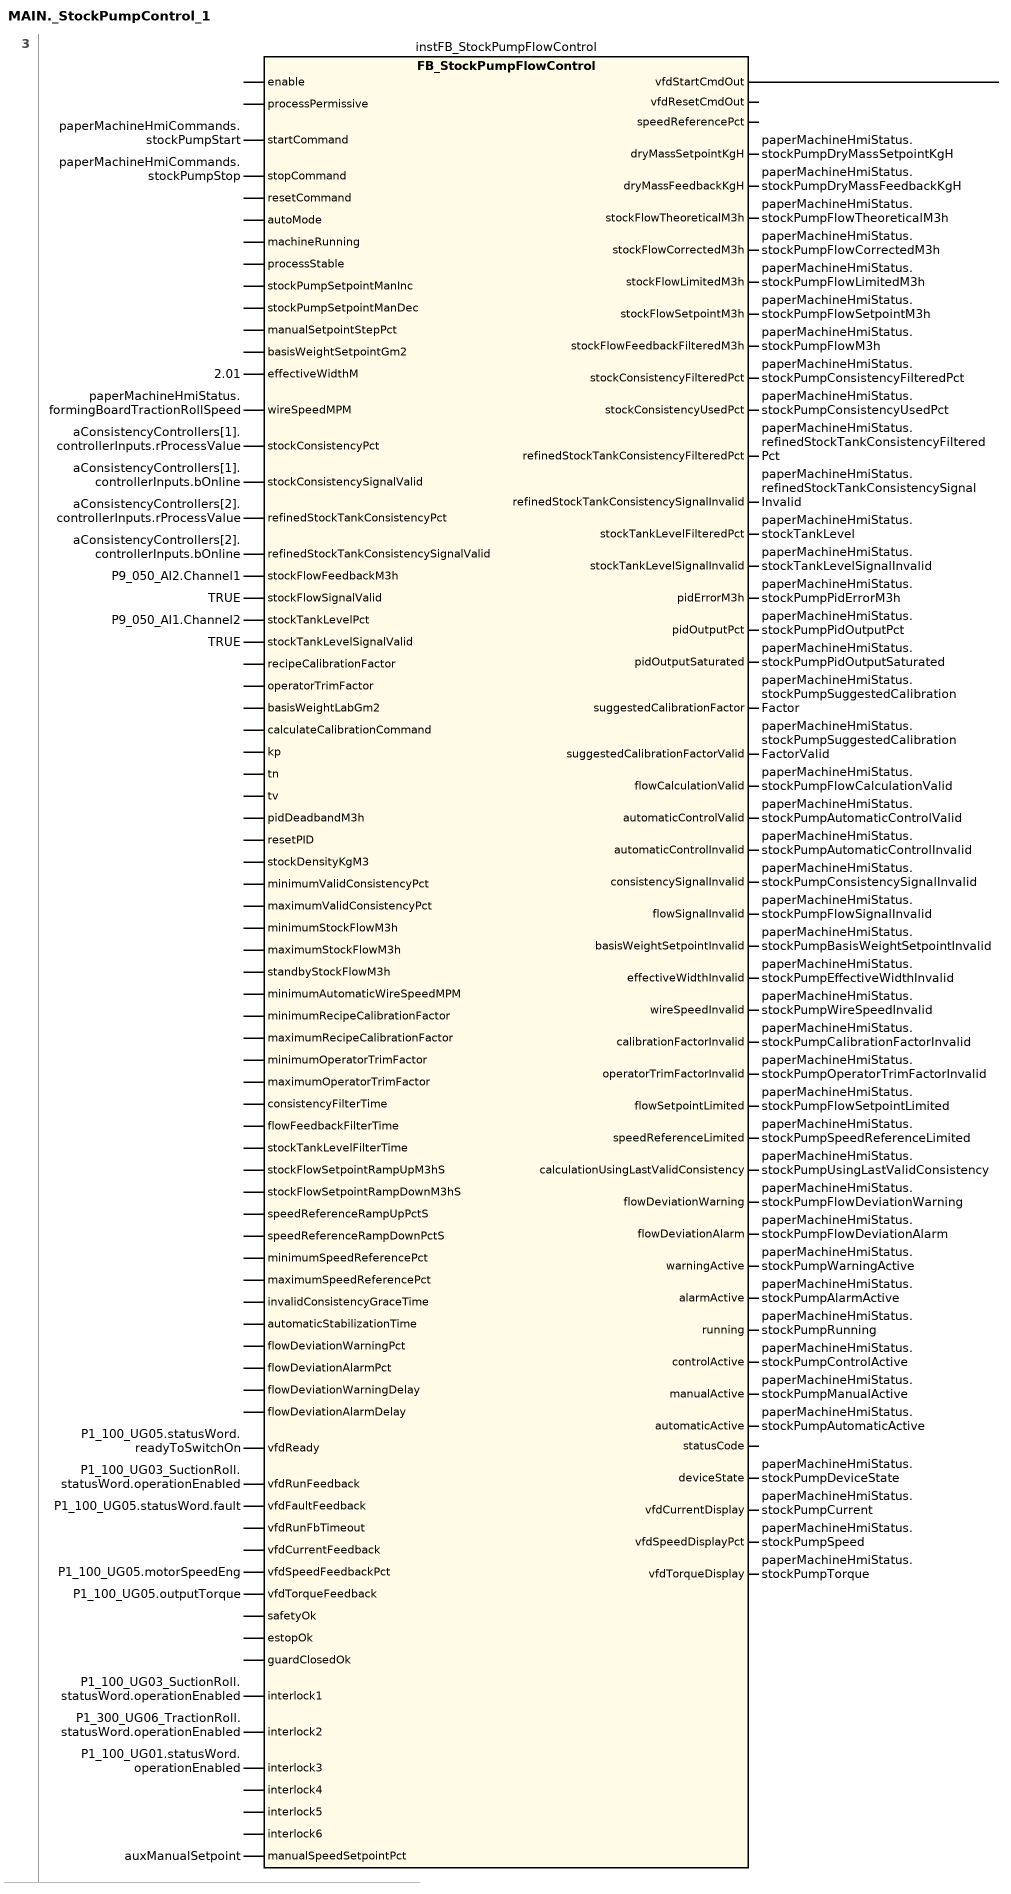
// NETWORK 3
instFB_StockPumpFlowControl(
    startCommand := paperMachineHmiCommands.stockPumpStart,
    stopCommand := paperMachineHmiCommands.stockPumpStop,
    effectiveWidthM := 2.01,
    wireSpeedMPM := paperMachineHmiStatus.formingBoardTractionRollSpeed,
    stockConsistencyPct := aConsistencyControllers[1].controllerInputs.rProcessValue,
    stockConsistencySignalValid := aConsistencyControllers[1].controllerInputs.bOnline,
    refinedStockTankConsistencyPct := aConsistencyControllers[2].controllerInputs.rProcessValue,
    refinedStockTankConsistencySignalValid := aConsistencyControllers[2].controllerInputs.bOnline,
    stockFlowFeedbackM3h := P9_050_AI2.Channel1,
    stockFlowSignalValid := TRUE,
    stockTankLevelPct := P9_050_AI1.Channel2,
    stockTankLevelSignalValid := TRUE,
    vfdReady := P1_100_UG05.statusWord.readyToSwitchOn,
    vfdRunFeedback := P1_100_UG03_SuctionRoll.statusWord.operationEnabled,
    vfdFaultFeedback := P1_100_UG05.statusWord.fault,
    vfdSpeedFeedbackPct := P1_100_UG05.motorSpeedEng,
    vfdTorqueFeedback := P1_100_UG05.outputTorque,
    interlock1 := P1_100_UG03_SuctionRoll.statusWord.operationEnabled,
    interlock2 := P1_300_UG06_TractionRoll.statusWord.operationEnabled,
    interlock3 := P1_100_UG01.statusWord.operationEnabled,
    manualSpeedSetpointPct := auxManualSetpoint,
    dryMassSetpointKgH => paperMachineHmiStatus.stockPumpDryMassSetpointKgH,
    dryMassFeedbackKgH => paperMachineHmiStatus.stockPumpDryMassFeedbackKgH,
    stockFlowTheoreticalM3h => paperMachineHmiStatus.stockPumpFlowTheoreticalM3h,
    stockFlowCorrectedM3h => paperMachineHmiStatus.stockPumpFlowCorrectedM3h,
    stockFlowLimitedM3h => paperMachineHmiStatus.stockPumpFlowLimitedM3h,
    stockFlowSetpointM3h => paperMachineHmiStatus.stockPumpFlowSetpointM3h,
    stockFlowFeedbackFilteredM3h => paperMachineHmiStatus.stockPumpFlowM3h,
    stockConsistencyFilteredPct => paperMachineHmiStatus.stockPumpConsistencyFilteredPct,
    stockConsistencyUsedPct => paperMachineHmiStatus.stockPumpConsistencyUsedPct,
    refinedStockTankConsistencyFilteredPct => paperMachineHmiStatus.refinedStockTankConsistencyFilteredPct,
    refinedStockTankConsistencySignalInvalid => paperMachineHmiStatus.refinedStockTankConsistencySignalInvalid,
    stockTankLevelFilteredPct => paperMachineHmiStatus.stockTankLevel,
    stockTankLevelSignalInvalid => paperMachineHmiStatus.stockTankLevelSignalInvalid,
    pidErrorM3h => paperMachineHmiStatus.stockPumpPidErrorM3h,
    pidOutputPct => paperMachineHmiStatus.stockPumpPidOutputPct,
    pidOutputSaturated => paperMachineHmiStatus.stockPumpPidOutputSaturated,
    suggestedCalibrationFactor => paperMachineHmiStatus.stockPumpSuggestedCalibrationFactor,
    suggestedCalibrationFactorValid => paperMachineHmiStatus.stockPumpSuggestedCalibrationFactorValid,
    flowCalculationValid => paperMachineHmiStatus.stockPumpFlowCalculationValid,
    automaticControlValid => paperMachineHmiStatus.stockPumpAutomaticControlValid,
    automaticControlInvalid => paperMachineHmiStatus.stockPumpAutomaticControlInvalid,
    consistencySignalInvalid => paperMachineHmiStatus.stockPumpConsistencySignalInvalid,
    flowSignalInvalid => paperMachineHmiStatus.stockPumpFlowSignalInvalid,
    basisWeightSetpointInvalid => paperMachineHmiStatus.stockPumpBasisWeightSetpointInvalid,
    effectiveWidthInvalid => paperMachineHmiStatus.stockPumpEffectiveWidthInvalid,
    wireSpeedInvalid => paperMachineHmiStatus.stockPumpWireSpeedInvalid,
    calibrationFactorInvalid => paperMachineHmiStatus.stockPumpCalibrationFactorInvalid,
    operatorTrimFactorInvalid => paperMachineHmiStatus.stockPumpOperatorTrimFactorInvalid,
    flowSetpointLimited => paperMachineHmiStatus.stockPumpFlowSetpointLimited,
    speedReferenceLimited => paperMachineHmiStatus.stockPumpSpeedReferenceLimited,
    calculationUsingLastValidConsistency => paperMachineHmiStatus.stockPumpUsingLastValidConsistency,
    flowDeviationWarning => paperMachineHmiStatus.stockPumpFlowDeviationWarning,
    flowDeviationAlarm => paperMachineHmiStatus.stockPumpFlowDeviationAlarm,
    warningActive => paperMachineHmiStatus.stockPumpWarningActive,
    alarmActive => paperMachineHmiStatus.stockPumpAlarmActive,
    running => paperMachineHmiStatus.stockPumpRunning,
    controlActive => paperMachineHmiStatus.stockPumpControlActive,
    manualActive => paperMachineHmiStatus.stockPumpManualActive,
    automaticActive => paperMachineHmiStatus.stockPumpAutomaticActive,
    deviceState => paperMachineHmiStatus.stockPumpDeviceState,
    vfdCurrentDisplay => paperMachineHmiStatus.stockPumpCurrent,
    vfdSpeedDisplayPct => paperMachineHmiStatus.stockPumpSpeed,
    vfdTorqueDisplay => paperMachineHmiStatus.stockPumpTorque); // FB_StockPumpFlowControl
END_METHOD

METHOD _VaccumPumps
VAR_INPUT
END_VAR
(*

    // ─────────────── LOW VACUUM EXHAUST FAN ───────────────
    lowVacuumExhaustFanStart : BOOL;  // Start low vacuum exhaust fan (Ligar exaustor do baixo vácuo)
    lowVacuumExhaustFanStop  : BOOL;  // Stop low vacuum exhaust fan (Parar exaustor do baixo vácuo)
	
	paperMachineHmiCommands.suctionRollVacuumPumpStart
	paperMachineHmiCommands.suctionRollVacuumPumpStop
	paperMachineHmiCommands.wireVacuumPumpStart
	paperMachineHmiCommands.wireVacuumPumpStop


*)
VAR_INST // added by the converter: edge detectors and wires of the graphical bodies
    _w1 : BOOL;
END_VAR
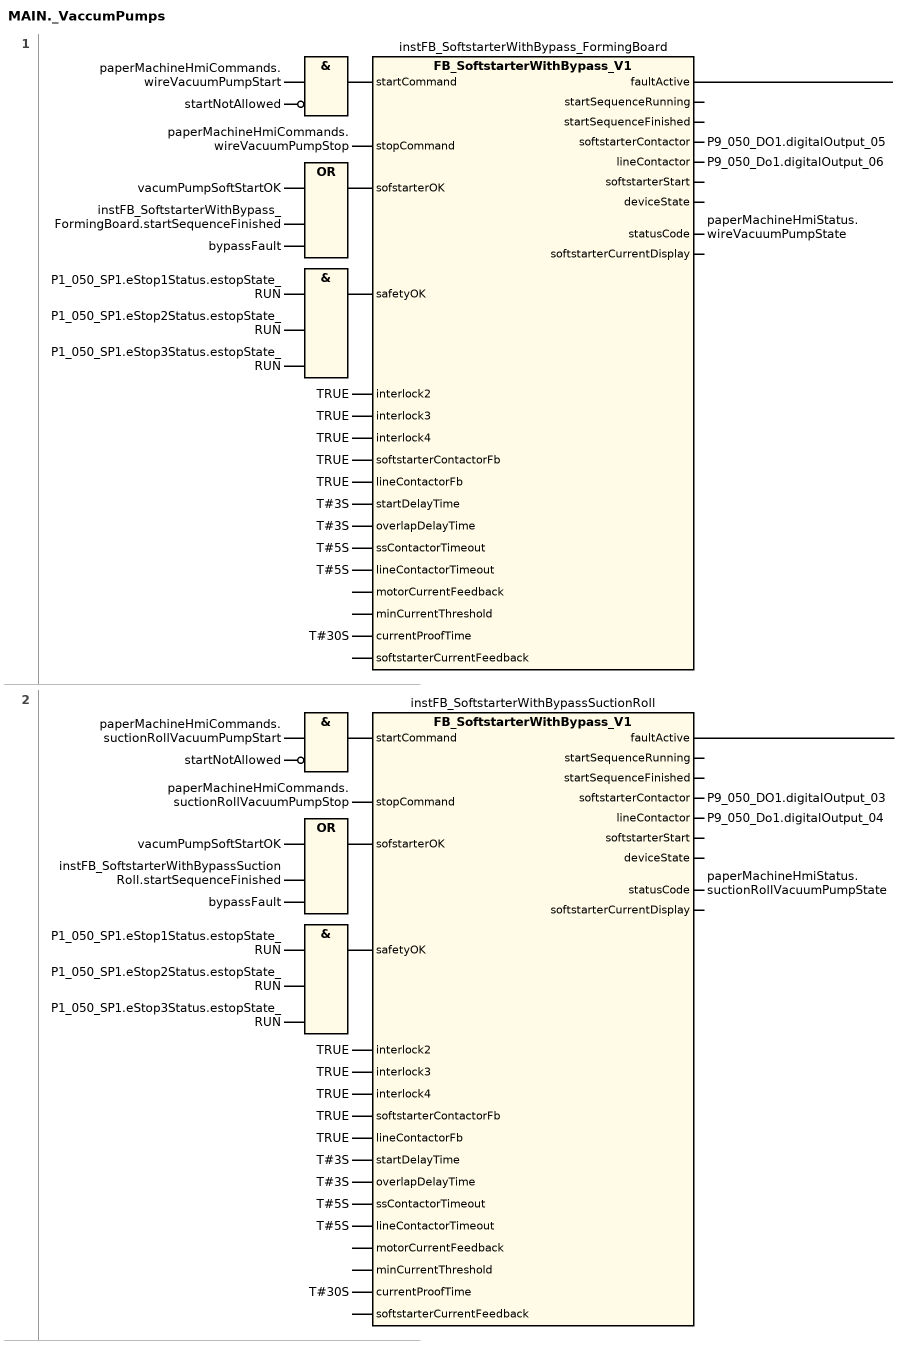
// NETWORK 1
instFB_SoftstarterWithBypass_FormingBoard(
    startCommand := paperMachineHmiCommands.wireVacuumPumpStart AND NOT startNotAllowed,
    stopCommand := paperMachineHmiCommands.wireVacuumPumpStop,
    sofstarterOK := vacumPumpSoftStartOK OR instFB_SoftstarterWithBypass_FormingBoard.startSequenceFinished OR bypassFault,
    safetyOK := P1_050_SP1.eStop1Status.estopState_RUN AND P1_050_SP1.eStop2Status.estopState_RUN AND P1_050_SP1.eStop3Status.estopState_RUN,
    interlock2 := TRUE,
    interlock3 := TRUE,
    interlock4 := TRUE,
    softstarterContactorFb := TRUE,
    lineContactorFb := TRUE,
    startDelayTime := T#3S,
    overlapDelayTime := T#3S,
    ssContactorTimeout := T#5S,
    lineContactorTimeout := T#5S,
    currentProofTime := T#30S,
    softstarterContactor => P9_050_DO1.digitalOutput_05,
    lineContactor => P9_050_Do1.digitalOutput_06,
    statusCode => paperMachineHmiStatus.wireVacuumPumpState); // FB_SoftstarterWithBypass_V1

// NETWORK 2
instFB_SoftstarterWithBypassSuctionRoll(
    startCommand := paperMachineHmiCommands.suctionRollVacuumPumpStart AND NOT startNotAllowed,
    stopCommand := paperMachineHmiCommands.suctionRollVacuumPumpStop,
    sofstarterOK := vacumPumpSoftStartOK OR instFB_SoftstarterWithBypassSuctionRoll.startSequenceFinished OR bypassFault,
    safetyOK := P1_050_SP1.eStop1Status.estopState_RUN AND P1_050_SP1.eStop2Status.estopState_RUN AND P1_050_SP1.eStop3Status.estopState_RUN,
    interlock2 := TRUE,
    interlock3 := TRUE,
    interlock4 := TRUE,
    softstarterContactorFb := TRUE,
    lineContactorFb := TRUE,
    startDelayTime := T#3S,
    overlapDelayTime := T#3S,
    ssContactorTimeout := T#5S,
    lineContactorTimeout := T#5S,
    currentProofTime := T#30S,
    softstarterContactor => P9_050_DO1.digitalOutput_03,
    lineContactor => P9_050_Do1.digitalOutput_04,
    statusCode => paperMachineHmiStatus.suctionRollVacuumPumpState); // FB_SoftstarterWithBypass_V1

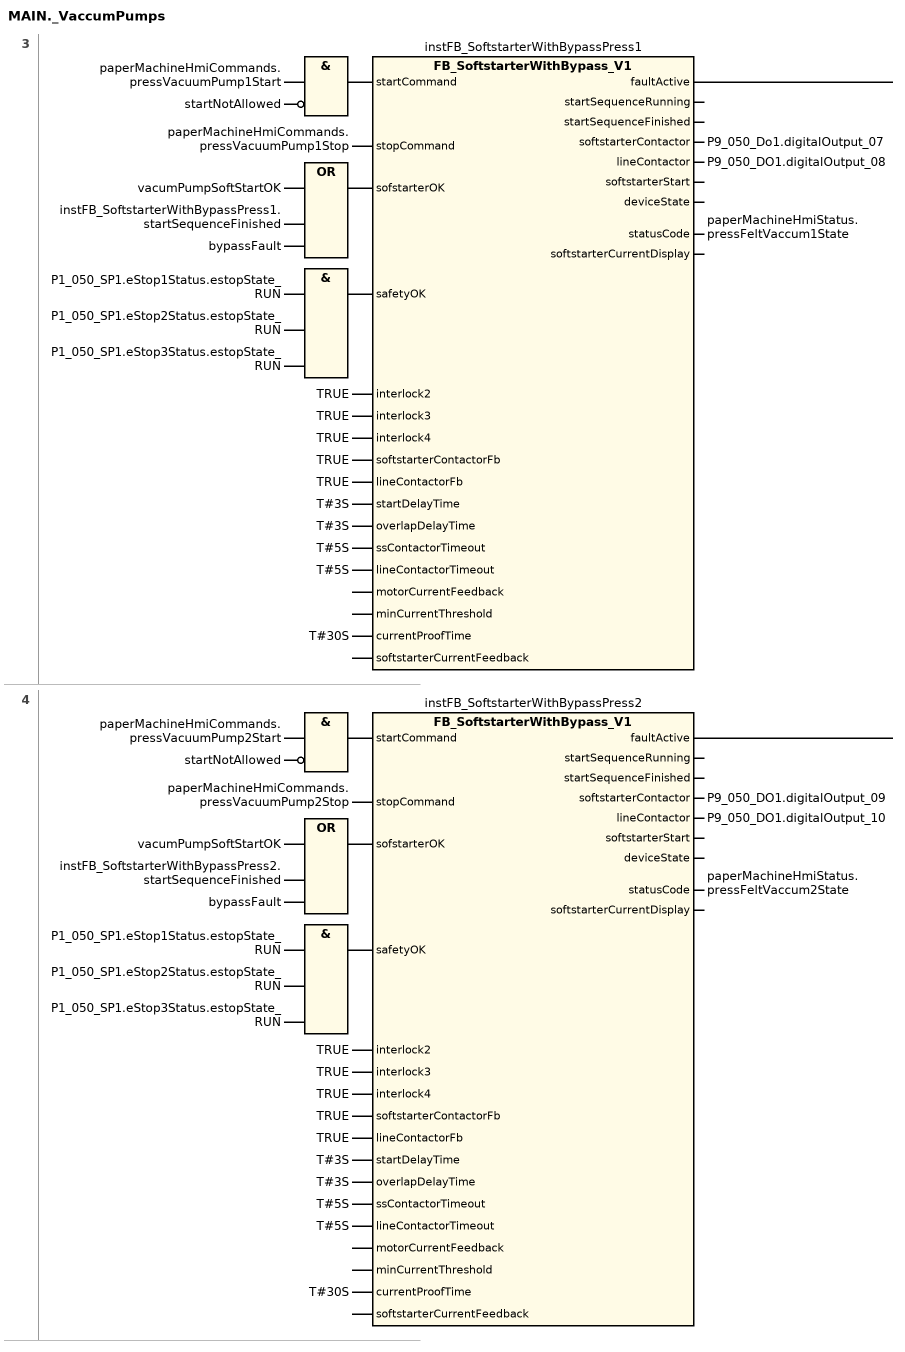
// NETWORK 3
instFB_SoftstarterWithBypassPress1(
    startCommand := paperMachineHmiCommands.pressVacuumPump1Start AND NOT startNotAllowed,
    stopCommand := paperMachineHmiCommands.pressVacuumPump1Stop,
    sofstarterOK := vacumPumpSoftStartOK OR instFB_SoftstarterWithBypassPress1.startSequenceFinished OR bypassFault,
    safetyOK := P1_050_SP1.eStop1Status.estopState_RUN AND P1_050_SP1.eStop2Status.estopState_RUN AND P1_050_SP1.eStop3Status.estopState_RUN,
    interlock2 := TRUE,
    interlock3 := TRUE,
    interlock4 := TRUE,
    softstarterContactorFb := TRUE,
    lineContactorFb := TRUE,
    startDelayTime := T#3S,
    overlapDelayTime := T#3S,
    ssContactorTimeout := T#5S,
    lineContactorTimeout := T#5S,
    currentProofTime := T#30S,
    softstarterContactor => P9_050_Do1.digitalOutput_07,
    lineContactor => P9_050_DO1.digitalOutput_08,
    statusCode => paperMachineHmiStatus.pressFeltVaccum1State); // FB_SoftstarterWithBypass_V1

// NETWORK 4
instFB_SoftstarterWithBypassPress2(
    startCommand := paperMachineHmiCommands.pressVacuumPump2Start AND NOT startNotAllowed,
    stopCommand := paperMachineHmiCommands.pressVacuumPump2Stop,
    sofstarterOK := vacumPumpSoftStartOK OR instFB_SoftstarterWithBypassPress2.startSequenceFinished OR bypassFault,
    safetyOK := P1_050_SP1.eStop1Status.estopState_RUN AND P1_050_SP1.eStop2Status.estopState_RUN AND P1_050_SP1.eStop3Status.estopState_RUN,
    interlock2 := TRUE,
    interlock3 := TRUE,
    interlock4 := TRUE,
    softstarterContactorFb := TRUE,
    lineContactorFb := TRUE,
    startDelayTime := T#3S,
    overlapDelayTime := T#3S,
    ssContactorTimeout := T#5S,
    lineContactorTimeout := T#5S,
    currentProofTime := T#30S,
    softstarterContactor => P9_050_DO1.digitalOutput_09,
    lineContactor => P9_050_DO1.digitalOutput_10,
    statusCode => paperMachineHmiStatus.pressFeltVaccum2State); // FB_SoftstarterWithBypass_V1

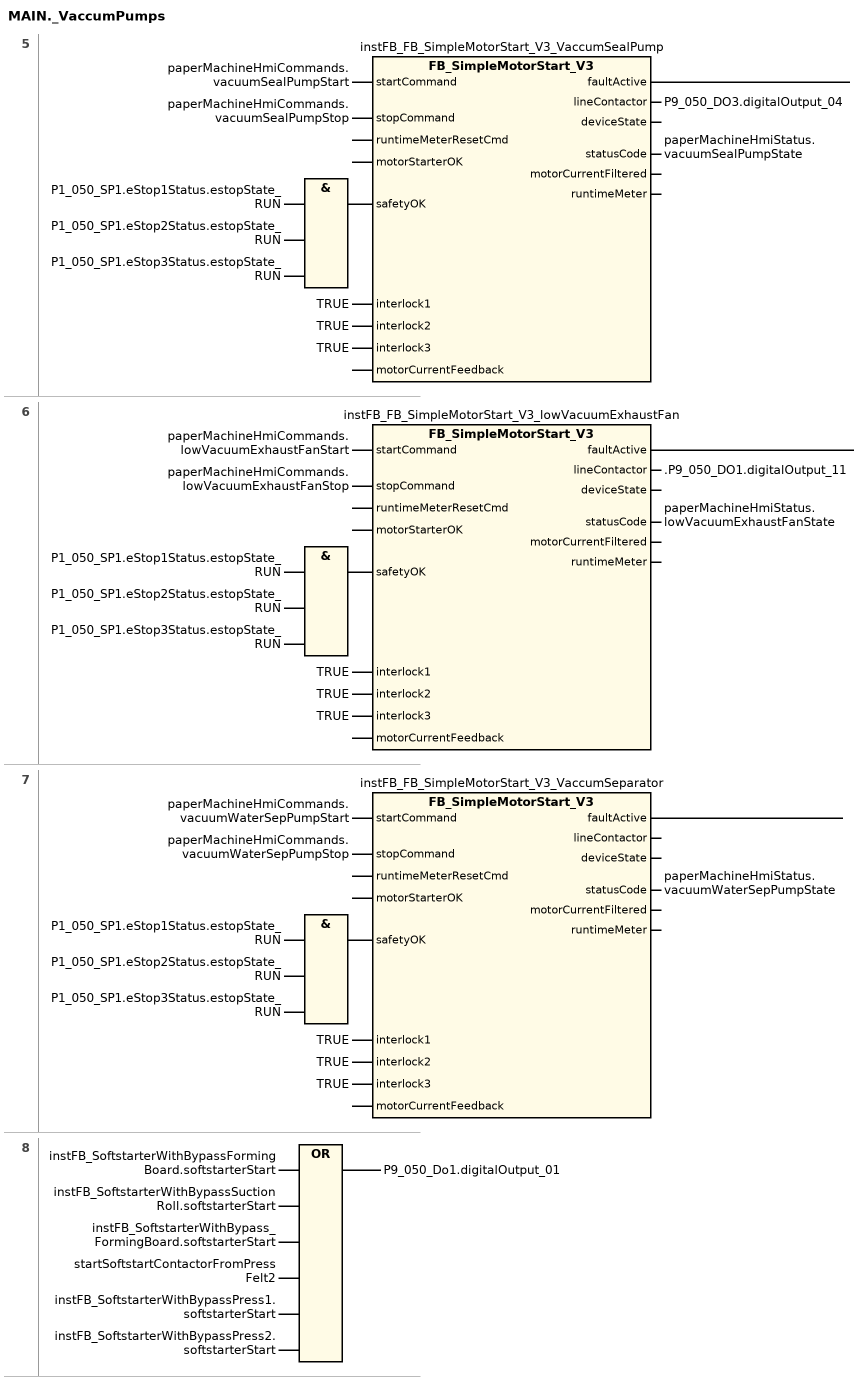
// NETWORK 5
instFB_FB_SimpleMotorStart_V3_VaccumSealPump(
    startCommand := paperMachineHmiCommands.vacuumSealPumpStart,
    stopCommand := paperMachineHmiCommands.vacuumSealPumpStop,
    safetyOK := P1_050_SP1.eStop1Status.estopState_RUN AND P1_050_SP1.eStop2Status.estopState_RUN AND P1_050_SP1.eStop3Status.estopState_RUN,
    interlock1 := TRUE,
    interlock2 := TRUE,
    interlock3 := TRUE,
    lineContactor => P9_050_DO3.digitalOutput_04,
    statusCode => paperMachineHmiStatus.vacuumSealPumpState); // FB_SimpleMotorStart_V3

// NETWORK 6
instFB_FB_SimpleMotorStart_V3_lowVacuumExhaustFan(
    startCommand := paperMachineHmiCommands.lowVacuumExhaustFanStart,
    stopCommand := paperMachineHmiCommands.lowVacuumExhaustFanStop,
    safetyOK := P1_050_SP1.eStop1Status.estopState_RUN AND P1_050_SP1.eStop2Status.estopState_RUN AND P1_050_SP1.eStop3Status.estopState_RUN,
    interlock1 := TRUE,
    interlock2 := TRUE,
    interlock3 := TRUE,
    lineContactor => .P9_050_DO1.digitalOutput_11,
    statusCode => paperMachineHmiStatus.lowVacuumExhaustFanState); // FB_SimpleMotorStart_V3

// NETWORK 7
instFB_FB_SimpleMotorStart_V3_VaccumSeparator(
    startCommand := paperMachineHmiCommands.vacuumWaterSepPumpStart,
    stopCommand := paperMachineHmiCommands.vacuumWaterSepPumpStop,
    safetyOK := P1_050_SP1.eStop1Status.estopState_RUN AND P1_050_SP1.eStop2Status.estopState_RUN AND P1_050_SP1.eStop3Status.estopState_RUN,
    interlock1 := TRUE,
    interlock2 := TRUE,
    interlock3 := TRUE,
    statusCode => paperMachineHmiStatus.vacuumWaterSepPumpState); // FB_SimpleMotorStart_V3

// NETWORK 8
P9_050_Do1.digitalOutput_01 := instFB_SoftstarterWithBypassFormingBoard.softstarterStart OR instFB_SoftstarterWithBypassSuctionRoll.softstarterStart OR instFB_SoftstarterWithBypass_FormingBoard.softstarterStart OR startSoftstartContactorFromPressFelt2 OR instFB_SoftstarterWithBypassPress1.softstarterStart OR instFB_SoftstarterWithBypassPress2.softstarterStart;

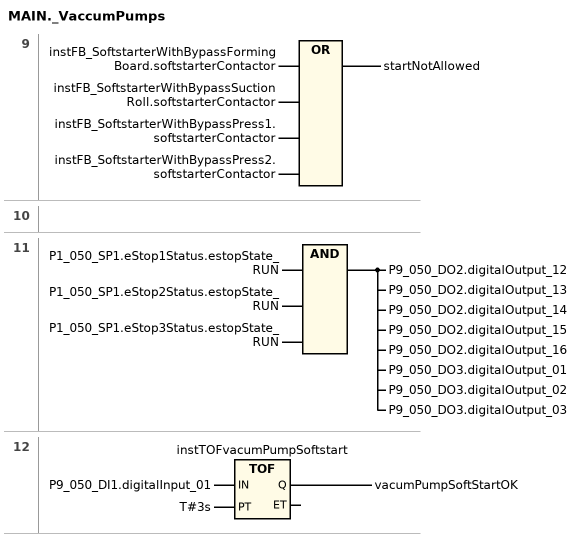
// NETWORK 9
startNotAllowed := instFB_SoftstarterWithBypassFormingBoard.softstarterContactor OR instFB_SoftstarterWithBypassSuctionRoll.softstarterContactor OR instFB_SoftstarterWithBypassPress1.softstarterContactor OR instFB_SoftstarterWithBypassPress2.softstarterContactor;

// NETWORK 10

// NETWORK 11
_w1 := P1_050_SP1.eStop1Status.estopState_RUN AND P1_050_SP1.eStop2Status.estopState_RUN AND P1_050_SP1.eStop3Status.estopState_RUN;
P9_050_DO2.digitalOutput_12 := _w1;
P9_050_DO2.digitalOutput_13 := _w1;
P9_050_DO2.digitalOutput_14 := _w1;
P9_050_DO2.digitalOutput_15 := _w1;
P9_050_DO2.digitalOutput_16 := _w1;
P9_050_DO3.digitalOutput_01 := _w1;
P9_050_DO3.digitalOutput_02 := _w1;
P9_050_DO3.digitalOutput_03 := _w1;

// NETWORK 12
instTOFvacumPumpSoftstart(IN := P9_050_DI1.digitalInput_01, PT := T#3s); // TOF
vacumPumpSoftStartOK := instTOFvacumPumpSoftstart.Q;
END_METHOD

METHOD _VaccumPumpWaterSeparator : BOOL
VAR_INPUT
END_VAR
(*

    vacuumWaterSepPumpStart  : BOOL;  // Start water separator vacuum pump (Ligar bomba de vácuo separadora de água)
    vacuumWaterSepPumpStop   : BOOL;  // Stop water separator vacuum pump (Parar bomba de vácuo separadora de água)
 	vacuumWaterSepAutoMan      : BOOL;  // Auto/manual mode select (Seleção automático/manual)
    vacuumWaterSepSetpointMan  : REAL;  // Manual setpoint (Setpoint manual)
    vacuumWaterSepSetpointAuto : REAL;  // Auto setpoint (Setpoint automático)	
	
*)
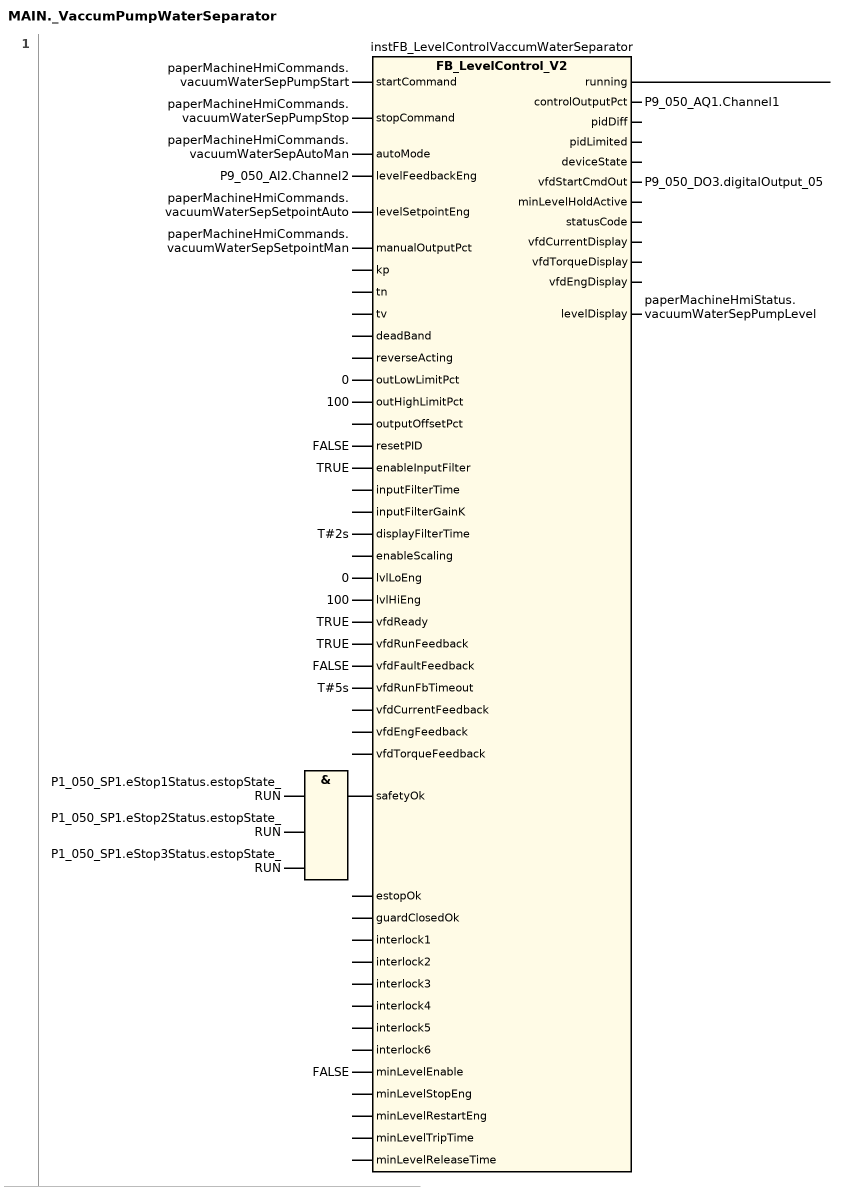
// NETWORK 1
instFB_LevelControlVaccumWaterSeparator(
    startCommand := paperMachineHmiCommands.vacuumWaterSepPumpStart,
    stopCommand := paperMachineHmiCommands.vacuumWaterSepPumpStop,
    autoMode := paperMachineHmiCommands.vacuumWaterSepAutoMan,
    levelFeedbackEng := P9_050_AI2.Channel2,
    levelSetpointEng := paperMachineHmiCommands.vacuumWaterSepSetpointAuto,
    manualOutputPct := paperMachineHmiCommands.vacuumWaterSepSetpointMan,
    outLowLimitPct := 0,
    outHighLimitPct := 100,
    resetPID := FALSE,
    enableInputFilter := TRUE,
    displayFilterTime := T#2s,
    lvlLoEng := 0,
    lvlHiEng := 100,
    vfdReady := TRUE,
    vfdRunFeedback := TRUE,
    vfdFaultFeedback := FALSE,
    vfdRunFbTimeout := T#5s,
    safetyOk := P1_050_SP1.eStop1Status.estopState_RUN AND P1_050_SP1.eStop2Status.estopState_RUN AND P1_050_SP1.eStop3Status.estopState_RUN,
    minLevelEnable := FALSE,
    controlOutputPct => P9_050_AQ1.Channel1,
    vfdStartCmdOut => P9_050_DO3.digitalOutput_05,
    levelDisplay => paperMachineHmiStatus.vacuumWaterSepPumpLevel); // FB_LevelControl_V2

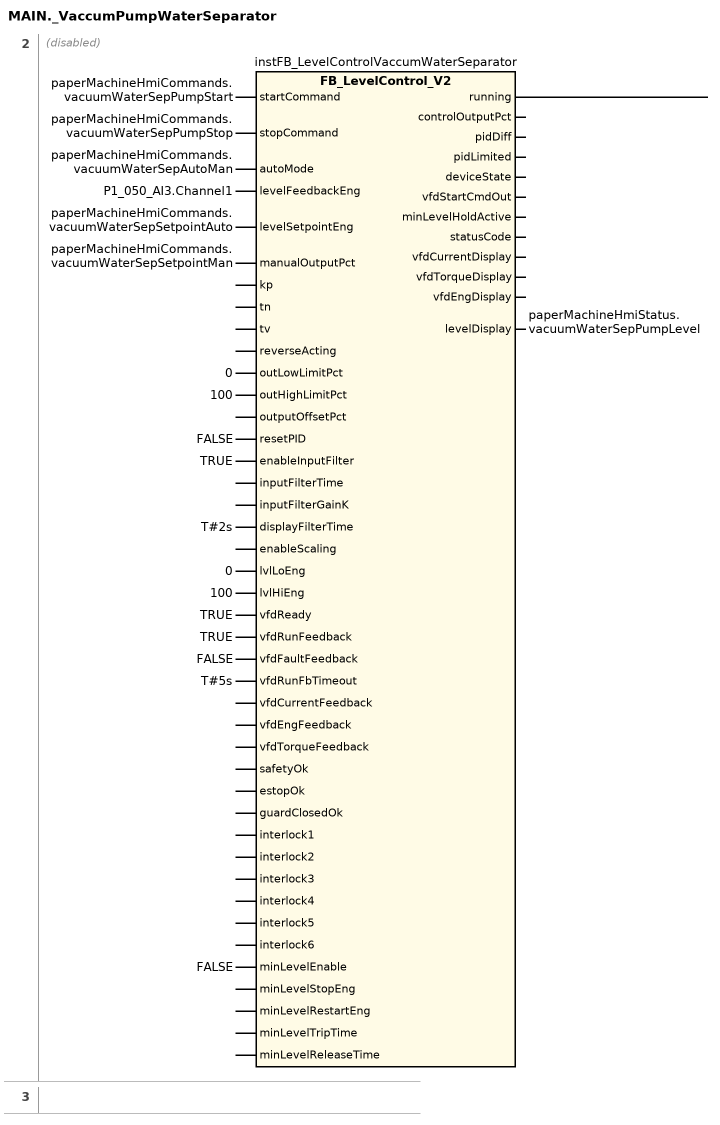
// NETWORK 2 (disabled)
// instFB_LevelControlVaccumWaterSeparator(
//     startCommand := paperMachineHmiCommands.vacuumWaterSepPumpStart,
//     stopCommand := paperMachineHmiCommands.vacuumWaterSepPumpStop,
//     autoMode := paperMachineHmiCommands.vacuumWaterSepAutoMan,
//     levelFeedbackEng := P1_050_AI3.Channel1,
//     levelSetpointEng := paperMachineHmiCommands.vacuumWaterSepSetpointAuto,
//     manualOutputPct := paperMachineHmiCommands.vacuumWaterSepSetpointMan,
//     outLowLimitPct := 0,
//     outHighLimitPct := 100,
//     resetPID := FALSE,
//     enableInputFilter := TRUE,
//     displayFilterTime := T#2s,
//     lvlLoEng := 0,
//     lvlHiEng := 100,
//     vfdReady := TRUE,
//     vfdRunFeedback := TRUE,
//     vfdFaultFeedback := FALSE,
//     vfdRunFbTimeout := T#5s,
//     minLevelEnable := FALSE,
//     levelDisplay => paperMachineHmiStatus.vacuumWaterSepPumpLevel); // FB_LevelControl_V2

// NETWORK 3
END_METHOD

METHOD _WirePitControl
VAR_INPUT
END_VAR
//P1_050_AI4.Channel1
(*

paperMachineHmiCommands.whiteWaterSiloSetpointMan
paperMachineHmiCommands.whiteWaterSiloSetpointAuto
paperMachineHmiCommands.wirePitSetpointMan
paperMachineHmiCommands.wirePitSetpointAuto
*)
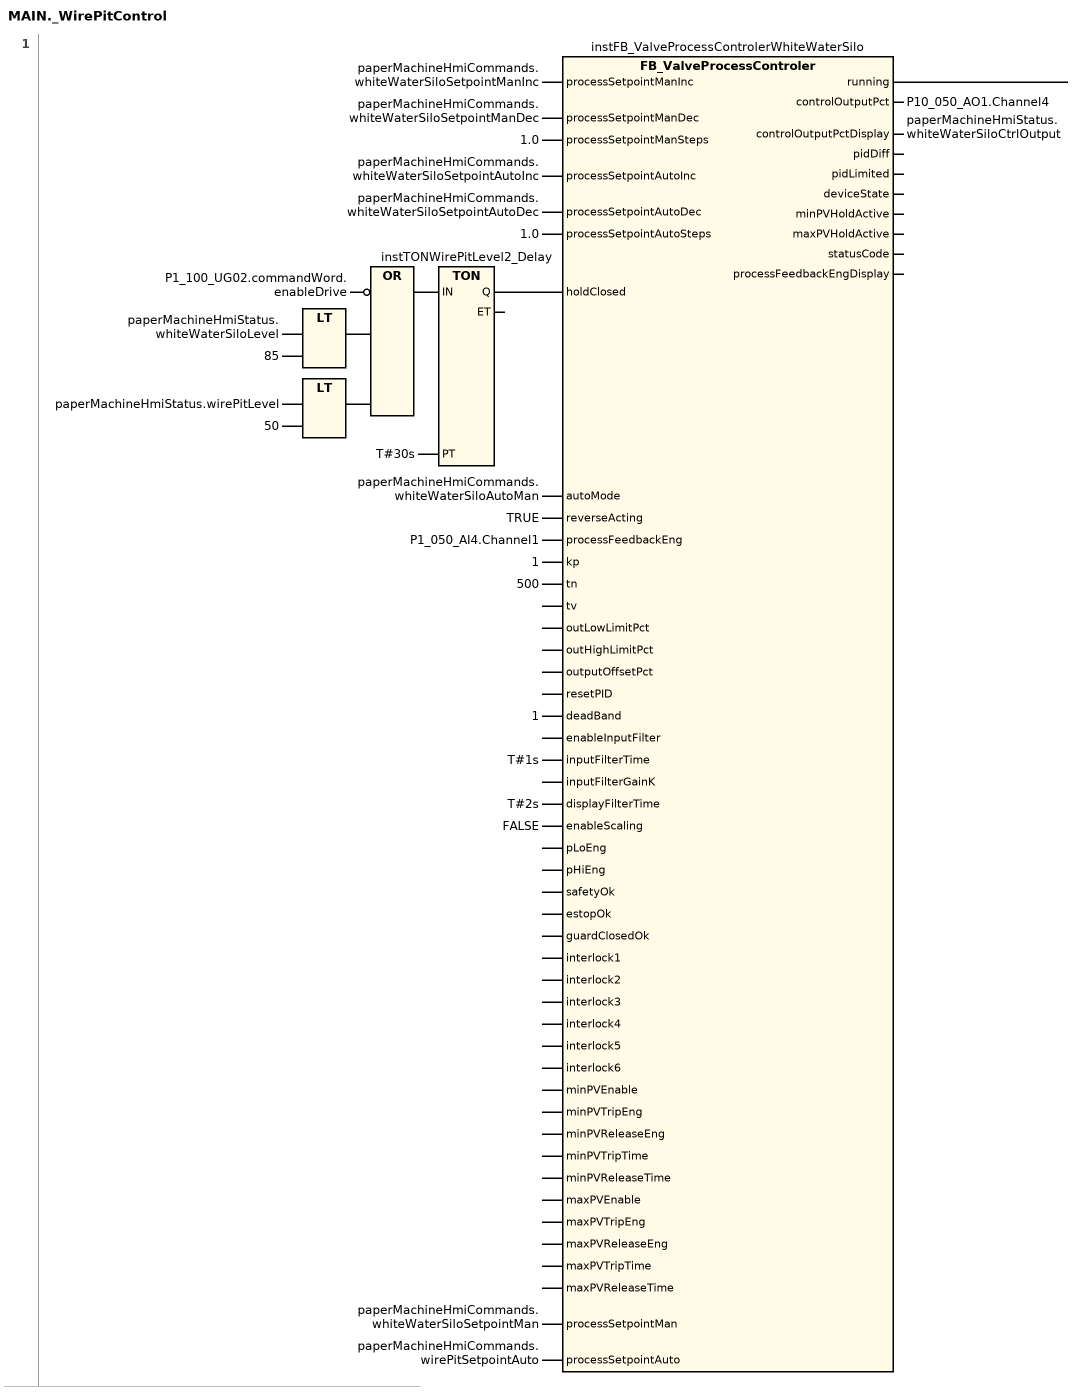
// NETWORK 1
instTONWirePitLevel2_Delay(IN := NOT P1_100_UG02.commandWord.enableDrive OR paperMachineHmiStatus.whiteWaterSiloLevel < 85 OR paperMachineHmiStatus.wirePitLevel < 50, PT := T#30s); // TON
instFB_ValveProcessControlerWhiteWaterSilo(
    processSetpointManInc := paperMachineHmiCommands.whiteWaterSiloSetpointManInc,
    processSetpointManDec := paperMachineHmiCommands.whiteWaterSiloSetpointManDec,
    processSetpointManSteps := 1.0,
    processSetpointAutoInc := paperMachineHmiCommands.whiteWaterSiloSetpointAutoInc,
    processSetpointAutoDec := paperMachineHmiCommands.whiteWaterSiloSetpointAutoDec,
    processSetpointAutoSteps := 1.0,
    holdClosed := instTONWirePitLevel2_Delay.Q,
    autoMode := paperMachineHmiCommands.whiteWaterSiloAutoMan,
    reverseActing := TRUE,
    processFeedbackEng := P1_050_AI4.Channel1,
    kp := 1,
    tn := 500,
    deadBand := 1,
    inputFilterTime := T#1s,
    displayFilterTime := T#2s,
    enableScaling := FALSE,
    processSetpointMan := paperMachineHmiCommands.whiteWaterSiloSetpointMan,
    processSetpointAuto := paperMachineHmiCommands.wirePitSetpointAuto,
    controlOutputPct => P10_050_AO1.Channel4,
    controlOutputPctDisplay => paperMachineHmiStatus.whiteWaterSiloCtrlOutput); // FB_ValveProcessControler

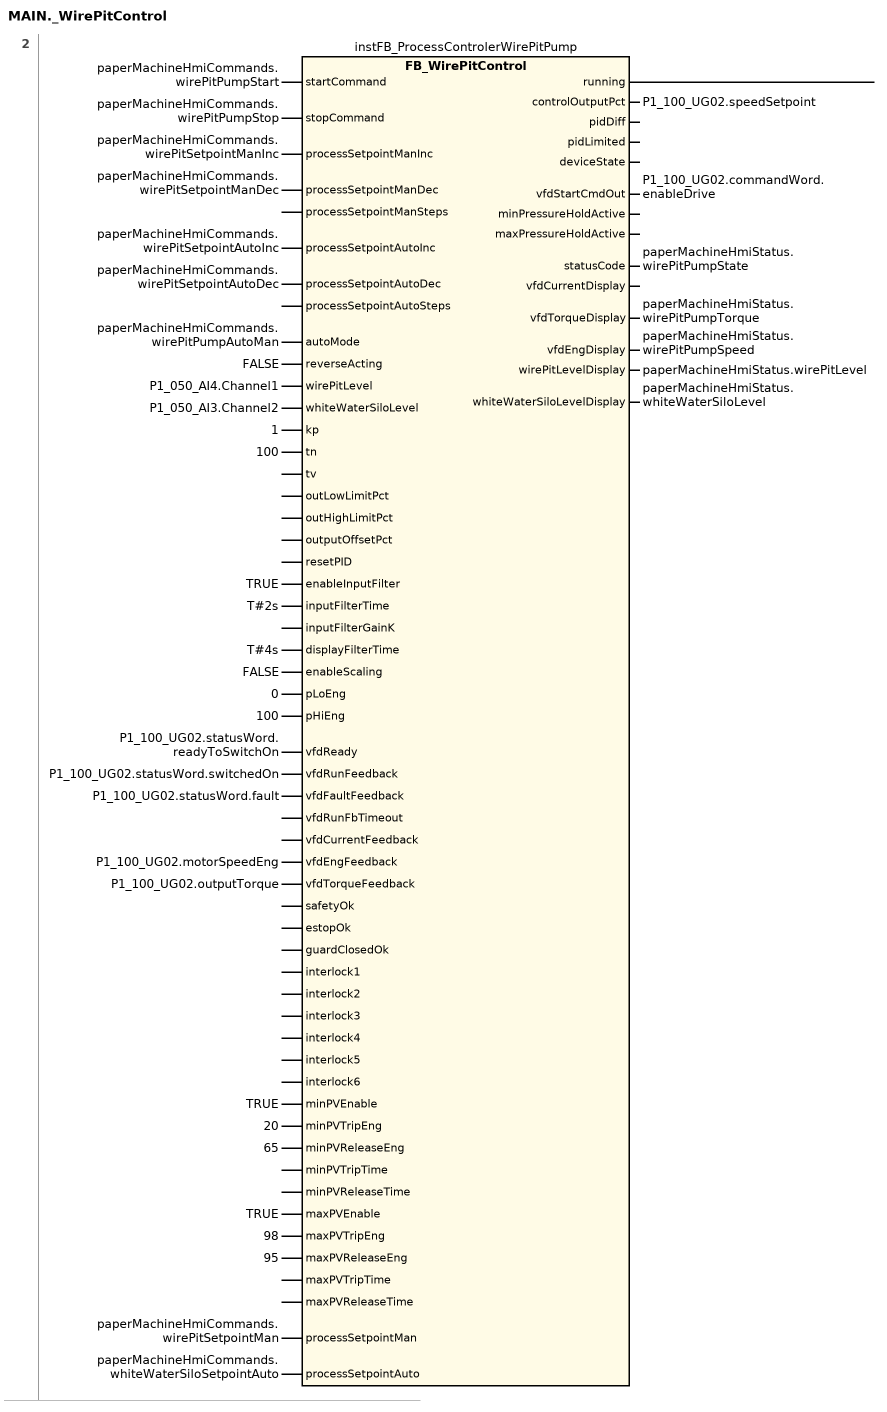
// NETWORK 2
instFB_ProcessControlerWirePitPump(
    startCommand := paperMachineHmiCommands.wirePitPumpStart,
    stopCommand := paperMachineHmiCommands.wirePitPumpStop,
    processSetpointManInc := paperMachineHmiCommands.wirePitSetpointManInc,
    processSetpointManDec := paperMachineHmiCommands.wirePitSetpointManDec,
    processSetpointAutoInc := paperMachineHmiCommands.wirePitSetpointAutoInc,
    processSetpointAutoDec := paperMachineHmiCommands.wirePitSetpointAutoDec,
    autoMode := paperMachineHmiCommands.wirePitPumpAutoMan,
    reverseActing := FALSE,
    wirePitLevel := P1_050_AI4.Channel1,
    whiteWaterSiloLevel := P1_050_AI3.Channel2,
    kp := 1,
    tn := 100,
    enableInputFilter := TRUE,
    inputFilterTime := T#2s,
    displayFilterTime := T#4s,
    enableScaling := FALSE,
    pLoEng := 0,
    pHiEng := 100,
    vfdReady := P1_100_UG02.statusWord.readyToSwitchOn,
    vfdRunFeedback := P1_100_UG02.statusWord.switchedOn,
    vfdFaultFeedback := P1_100_UG02.statusWord.fault,
    vfdEngFeedback := P1_100_UG02.motorSpeedEng,
    vfdTorqueFeedback := P1_100_UG02.outputTorque,
    minPVEnable := TRUE,
    minPVTripEng := 20,
    minPVReleaseEng := 65,
    maxPVEnable := TRUE,
    maxPVTripEng := 98,
    maxPVReleaseEng := 95,
    processSetpointMan := paperMachineHmiCommands.wirePitSetpointMan,
    processSetpointAuto := paperMachineHmiCommands.whiteWaterSiloSetpointAuto,
    controlOutputPct => P1_100_UG02.speedSetpoint,
    vfdStartCmdOut => P1_100_UG02.commandWord.enableDrive,
    statusCode => paperMachineHmiStatus.wirePitPumpState,
    vfdTorqueDisplay => paperMachineHmiStatus.wirePitPumpTorque,
    vfdEngDisplay => paperMachineHmiStatus.wirePitPumpSpeed,
    wirePitLevelDisplay => paperMachineHmiStatus.wirePitLevel,
    whiteWaterSiloLevelDisplay => paperMachineHmiStatus.whiteWaterSiloLevel); // FB_WirePitControl
END_METHOD

METHOD machineReset
VAR_INPUT
END_VAR

VAR
	instTP_Reset: TP;
END_VAR
//────────────────────────────────────────────
// UG01 to UG06 (General Utilities / Aux Drives)
//────────────────────────────────────────────
P1_100_UG01.commandWord.faultResetCmd := paperMachineHmiCommands.machineReset;
P1_100_UG02.commandWord.faultResetCmd := paperMachineHmiCommands.machineReset;
P1_100_UG03_SuctionRoll.commandWord.faultResetCmd := paperMachineHmiCommands.machineReset;
P1_100_UG04.commandWord.faultResetCmd := paperMachineHmiCommands.machineReset;
P1_100_UG05.commandWord.faultResetCmd := paperMachineHmiCommands.machineReset;
P1_300_UG06_TractionRoll.commandWord.faultResetCmd := paperMachineHmiCommands.machineReset;

//────────────────────────────────────────────
// Safety PLC Reset
//────────────────────────────────────────────
P1_050_SP1.safetyReset := paperMachineHmiCommands.machineReset;
P1_050_SP1.errorAcknowledgement := paperMachineHmiCommands.machineReset;

//────────────────────────────────────────────
// Press Section Drives
//────────────────────────────────────────────
P11_400_UG01_SecondPress.commandWord.faultResetCmd := paperMachineHmiCommands.machineReset;
P12_400_UG01_FirstPress.commandWord.faultResetCmd := paperMachineHmiCommands.machineReset;

//────────────────────────────────────────────
// Drying Section — Group 1
//────────────────────────────────────────────
P13_500_UG01_1GR_UpperSlave.commandWord.faultResetCmd := paperMachineHmiCommands.machineReset;
P13_500_UG02_1GR_LowerMaster.commandWord.faultResetCmd := paperMachineHmiCommands.machineReset;
P13_500_UG03_1GR_UpperMaster.commandWord.faultResetCmd := paperMachineHmiCommands.machineReset;

//────────────────────────────────────────────
// Drying Section — Group 2
//────────────────────────────────────────────
P13_501_UG01_2GR_LowerSlave.commandWord.faultResetCmd := paperMachineHmiCommands.machineReset;
P13_501_UG02_2GR_UpperSlave.commandWord.faultResetCmd := paperMachineHmiCommands.machineReset;
P13_501_UG03_2GR_LowerMaster.commandWord.faultResetCmd := paperMachineHmiCommands.machineReset;
P14_501_UG01_2GR_UpperMaster.commandWord.faultResetCmd := paperMachineHmiCommands.machineReset;

//────────────────────────────────────────────
// Drying Section — Group 3
//────────────────────────────────────────────
P14_502_UG01_3GR_LowerSlave.commandWord.faultResetCmd := paperMachineHmiCommands.machineReset;
P14_502_UG02_3GR_UpperSlave.commandWord.faultResetCmd := paperMachineHmiCommands.machineReset;
P14_502_UG03_3GR_LowerMaster.commandWord.faultResetCmd := paperMachineHmiCommands.machineReset;
P14_502_UG04_3GR_UpperMaster.commandWord.faultResetCmd := paperMachineHmiCommands.machineReset;

//────────────────────────────────────────────
// Rewinder
//────────────────────────────────────────────
P15_600_UG01_Rewinder.commandWord.faultResetCmd := paperMachineHmiCommands.machineReset;
END_METHOD

END_PROGRAM

(* stored: Version 1.1.0.1, ProductVersion 3.1.4024.15
   POU MAIN: Id {5655f915-5dcf-4c87-91ff-2912e5ed07e4}, SpecialFunc None
   Method _000_Init_Variables: Id {5375a803-7613-4982-b9a2-f469ce258019}
   Method _001_FirstScan: Id {2b51631a-b1de-4251-88c9-0f83eb7f4089}
   Method _100_FormingBoardControl: Id {0c14a096-ab0f-45c1-953f-c1b000dd222b}
   Method _110_FormingBoardAux: Id {5aa4fd0c-47a3-4984-9a55-af92e2ae98ef}
   Method _200_PressSectionControl: Id {9f824a2c-9679-4031-8e2d-18b1073be726}
   Method _500_DryingSectionGroup1DriveControl: Id {7943a74e-10ea-458b-9502-2d49d50c4e35}
   Method _501_DryingSectionGroup2DriveControl: Id {f83f4d32-fa55-425e-9a54-fabf3c551fc1}
   Method _502_DryingSectionGroup3DriveControl: Id {9a974028-0ff1-4fc6-ae78-595db97cb730}
   Method _550_DryingSectionLubrification: Id {1c3ab415-b9c8-4039-a58e-5404ebefb0b7}
   Method _600_WinderGroup: Id {603ff0d1-31e4-4576-a200-a1a15c654d7f}
   Method _700_JumboWeightCapture: Id {91b550a2-c25c-4ad4-8451-18f91a23a77c}
   Method _750_ConsistencyControllersRead: Id {7bbace23-8b7c-4043-91cf-313a9c010b9f}
   Method _888_Alarms: Id {d9864b94-8b87-40be-9edc-0758f89dc5b9}
   Method _900_DriveFaultDiagnostics: Id {a7232a3a-7045-4ad4-87db-050a923ee00e}
   Method _CentrifugalPressureScreenControl: Id {18b0f911-c9ca-4b47-826f-de0cd0c5db50}
   Method _CouchPitMixerControl: Id {98f7283d-3c51-4c62-91d0-f4e2606ab671}
   Method _CouchPitPumpControl: Id {60edba15-dfcb-4145-807a-b545f9976fa8}
   Method _FunctionBlockTest: Id {dc68dec4-b8e1-4e42-9c46-f76b6e3f7d02}
   Method _HeadBoxAuxiliaryControls: Id {b4d5fe16-43ef-431f-9e3b-d46cb5910730}
   Method _MixPumpControl_1: Id {d62a7ec7-6a8b-4696-bc00-270cd3d733f9}
   Method _StockPumpControl: Id {44ec4fcc-2a75-4e83-963c-b807cac52e25}
   Method _StockPumpControl_1: Id {f30519d5-f949-4cda-b919-d3c5e6fdcad4}
   Method _VaccumPumps: Id {8d03af37-1f90-4067-bf6c-04d0e3d98f21}
   Method _VaccumPumpWaterSeparator: Id {6760ec0a-00ff-42af-9a64-01147fda43cf}
   Method _WirePitControl: Id {7d4a518b-870d-4ab9-a21a-ca0bad9abb45}
   Method machineReset: Id {02d7d166-7912-45b0-ae8c-bd34367b2eb6} *)
